// TIA Portal V15 export
// export: Created 2018-05-29T12:25:38.1552518Z, ExportSetting WithDefaults, DisplayName Totally Integrated Automation Portal, DisplayVersion V15, DisplayName TIA Portal Openness, DisplayVersion V15, DisplayName STEP 7 Professional, DisplayVersion V15, DisplayName WinCC Professional, DisplayVersion V15
FUNCTION "Equipment_Modules" : Void   // FC1, STL
TITLE = Program
{ S7_Optimized_Access := 'TRUE' }
VERSION : 0.1
// Call all the Equipment Modules
// stored: AutoNumber true, UDAEnableTagReadback false
BEGIN

NETWORK
TITLE = Main
// comment
	CALL	EM_Instance_1_fc
	CALL	EM_Instance_2_fc
	CALL	EM_Instance_3_fc
	CALL	EM_Instance_4_fc
	CALL	EM_Instance_5_fc
	CALL	EM_Instance_6_fc
	CALL	EM_Instance_7_fc
	CALL	EM_Instance_8_fc
	CALL	EM_Instance_9_fc
	CALL	EM_Instance_10_fc
	CALL	EM_Instance_11_fc
	CALL	EM_Instance_12_fc
	CALL	EM_Instance_13_fc
	CALL	EM_Instance_14_fc
END_FUNCTION
